FUNCTION F_QuatRotateVec3Point : FB_Vec3
VAR_INPUT
    iQuat : I_Quat;
    iVec3 : I_Vec3;
END_VAR
VAR_OUTPUT
    bError : BOOL;
    sErrorMsg : T_MaxString;
END_VAR
VAR
    fbQ : FB_Quaternion;
    fbV : FB_Vec3;
    fbQc : FB_Quaternion;
    fbQv : FB_Quaternion;
END_VAR


bError := FALSE;
sErrorMsg := '';

fbQ.Set(iQuat.w, iQuat.x, iQuat.y, iQuat.z);

IF fbQ.GetNorm() = 0.0 THEN
    bError := TRUE;
    sErrorMsg := 'Error: cannot rotate a vector using a quaternion with a norm of 0.';
    F_QuatRotateVec3Point.Set(iVec3.x, iVec3.y, iVec3.z);
    RETURN;
END_IF

fbQ.Normalize();

fbV.Set(iVec3.x, iVec3.y, iVec3.z);

fbQc := fbQ;
fbQc.MakeConj();

fbQv := F_MulQuat(fbQ, fbV);
fbQv := F_MulQuat(fbQv, fbQc);

F_QuatRotateVec3Point.Set(fbQv.x, fbQv.y, fbQv.z);

END_FUNCTION

(* stored: Version 1.1.0.1
   POU F_QuatRotateVec3Point: Id {6fce307e-53c6-4581-b61f-d13df4766960}, SpecialFunc None *)
